PROGRAM PRG_Output

VAR
	fbValveOutput : FB_ValveControl;
END_VAR

G_Enables.bEnableU := G_Mode.bRunning; // Lagt til senere

// Runs FB with given values
fbValveOutput(
	fNormalizedInput := G_OPC.fU,		// Signal to set spool at wanted position
	bEnable := G_Enables.bEnableU,		// Enable signal
	nOutput => G_Output.nValveOutput	// Output signal to valve
);

// If system is running, set green and red light on controller true. False when not running:
G_Output.bGreenLight := G_Mode.bRunning;
G_Output.bRedLight   := G_Mode.bRunning;

END_PROGRAM

(* stored: Version 1.1.0.1
   POU PRG_Output: Id {570651de-6d72-48ad-99bb-75936a9676a8}, SpecialFunc None *)
